TYPE ST_System_DLK_Zustand :
STRUCT
	Betrieb_Anford			: BOOL;
	Betrieb_Soll			: BOOL;
	Betrieb					: BOOL;

	Netze_Anford			: ST_Zustand_Netze_Anford;

	Freigabe				: BOOL;
	Freigabe_Deakt			: BOOL;
	Freigabe_Code			: WORD;

	Stoerung				: BOOL;
	Stoerung_Code			: WORD;

	Warnung					: BOOL;
	Warnung_Code			: WORD;

	Status					: SINT;
	Status_Vorl_Regelventil		: BOOL;
	Status_Vorl_Pumpe		: BOOL;
	Status_Nachl_Regelventil	: BOOL;
	Status_Nachl_Pumpe		: BOOL;

	Quittierung				: BOOL;

	Netz_WW_Anford			: ST_Zustand_Netz_Anford;

END_STRUCT
END_TYPE

(* stored: Version 1.1.0.1, ProductVersion 3.1.4024.9
   DUT ST_System_DLK_Zustand: Id {df6257e2-0812-4079-ba71-28497afb0024} *)
